(* IEC 61131-3 sources: vertical-injection-machine-docs/docs/IM_SYS_PRG/Code/IO管理/数字量输入, 3 files *)

(* ---- FB_PLCDigitalInputBinder.st ---- *)
(*
  FB_PLCDigitalInputBinder 功能块
  功能：
  1. 把 PLC 运行时输入映像 `IN[0..47]` 刷新到原始 IO 边界 `ST_PLCIO.X*`。
  2. 当前块只负责“采集现场原始数字量输入”，不直接转换为 `ST_MachineSensor`、`ST_PanelIO` 或其他工艺语义。
  3. 当前输入点位顺序固定按现场 IO 表绑定，若现场扩点或换点，必须同步修改本块和 `ST_PLCIO`。

  使用限制：
  1. 当前实现假定目标 PLC 运行时直接提供 `IN[]` 输入映像数组。
  2. 本块应在 `PRG_MainControl` 每拍最前段调用，确保后续逻辑消费到的是本拍最新原始输入。
*)
FUNCTION_BLOCK FB_PLCDigitalInputBinder
VAR_IN_OUT
    stPLC: ST_PLCIO; // 原始 PLC IO 共享边界；本块把现场 `IN[]` 输入映像逐点刷新到其中的 `X*` 字段。
END_VAR

stPLC.X0 := IN[0];      // 把 `IN[0]` 刷新到 `X0`，表示紧急回升原始输入。
stPLC.X1 := IN[1];      // 把 `IN[1]` 刷新到 `X1`，表示低压合模原始输入。
stPLC.X2 := IN[2];      // 把 `IN[2]` 刷新到 `X2`，表示高压合模原始输入。
stPLC.X3 := IN[3];      // 把 `IN[3]` 刷新到 `X3`，表示合模停止原始输入。
stPLC.X4 := IN[4];      // 把 `IN[4]` 刷新到 `X4`，表示电眼输入原始输入。
stPLC.X5 := IN[5];      // 把 `IN[5]` 刷新到 `X5`，表示储料停止原始输入。
stPLC.X6 := IN[6];      // 把 `IN[6]` 刷新到 `X6`，表示拉带停原始输入。
stPLC.X7 := IN[7];      // 把 `IN[7]` 刷新到 `X7`，表示拉带慢速原始输入。
stPLC.X10 := IN[8];     // 把 `IN[8]` 刷新到 `X10`，表示左合模原始输入。
stPLC.X11 := IN[9];     // 把 `IN[9]` 刷新到 `X11`，表示右合模原始输入。
stPLC.X12 := IN[10];    // 把 `IN[10]` 刷新到 `X12`，表示开模停止原始输入。
stPLC.X13 := IN[11];    // 把 `IN[11]` 刷新到 `X13`，表示左托进停原始输入。
stPLC.X14 := IN[12];    // 把 `IN[12]` 刷新到 `X14`，表示左托退停原始输入。
stPLC.X15 := IN[13];    // 把 `IN[13]` 刷新到 `X15`，表示倒带停原始输入。
stPLC.X16 := IN[14];    // 把 `IN[14]` 刷新到 `X16`，表示跳带停原始输入。
stPLC.X17 := IN[15];    // 把 `IN[15]` 刷新到 `X17`，表示二级射出原始输入。
stPLC.X20 := IN[16];    // 把 `IN[16]` 刷新到 `X20`，表示右托进停原始输入。
stPLC.X21 := IN[17];    // 把 `IN[17]` 刷新到 `X21`，表示右托退停原始输入。
stPLC.X22 := IN[18];    // 把 `IN[18]` 刷新到 `X22`，表示座退停止原始输入。
stPLC.X23 := IN[19];    // 把 `IN[19]` 刷新到 `X23`，表示座进停止原始输入。
stPLC.X24 := IN[20];    // 把 `IN[20]` 刷新到 `X24`，表示三级射出原始输入。
stPLC.X25 := IN[21];    // 把 `IN[21]` 刷新到 `X25`，表示中子进停原始输入。
stPLC.X26 := IN[22];    // 把 `IN[22]` 刷新到 `X26`，表示中子退停原始输入。
stPLC.X27 := IN[23];    // 把 `IN[23]` 刷新到 `X27`，表示马达故障原始输入。
stPLC.X30 := IN[24];    // 把 `IN[24]` 刷新到 `X30`，表示安全门原始输入。
stPLC.X31 := IN[25];    // 把 `IN[25]` 刷新到 `X31`，表示模具区域原始输入。
stPLC.X32 := IN[26];    // 把 `IN[26]` 刷新到 `X32`，表示机械手合模原始输入。
stPLC.X33 := IN[27];    // 把 `IN[27]` 刷新到 `X33`，表示机械手托模原始输入。
stPLC.X34 := IN[28];    // 把 `IN[28]` 刷新到 `X34`，表示备用原始输入。
stPLC.X35 := IN[29];    // 把 `IN[29]` 刷新到 `X35`，表示备用原始输入。
stPLC.X36 := IN[30];    // 把 `IN[30]` 刷新到 `X36`，表示射出停止原始输入。
stPLC.X37 := IN[31];    // 把 `IN[31]` 刷新到 `X37`，表示备用原始输入。
stPLC.X40 := IN[32];    // 把 `IN[32]` 刷新到 `X40`，表示备用原始输入。
stPLC.X41 := IN[33];    // 把 `IN[33]` 刷新到 `X41`，表示备用原始输入。
stPLC.X42 := IN[34];    // 把 `IN[34]` 刷新到 `X42`，表示备用原始输入。
stPLC.X43 := IN[35];    // 把 `IN[35]` 刷新到 `X43`，表示备用原始输入。
stPLC.X44 := IN[36];    // 把 `IN[36]` 刷新到 `X44`，表示备用原始输入。
stPLC.X45 := IN[37];    // 把 `IN[37]` 刷新到 `X45`，表示备用原始输入。
stPLC.X46 := IN[38];    // 把 `IN[38]` 刷新到 `X46`，表示备用原始输入。
stPLC.X47 := IN[39];    // 把 `IN[39]` 刷新到 `X47`，表示备用原始输入。
stPLC.X50 := IN[40];    // 把 `IN[40]` 刷新到 `X50`，当前暂定表示启动命令原始输入。
stPLC.X51 := IN[41];    // 把 `IN[41]` 刷新到 `X51`，当前暂定表示停止命令原始输入。
stPLC.X52 := IN[42];    // 把 `IN[42]` 刷新到 `X52`，当前暂定表示复位命令原始输入。
stPLC.X53 := IN[43];    // 把 `IN[43]` 刷新到 `X53`，当前暂定表示急停命令原始输入。
stPLC.X54 := IN[44];    // 把 `IN[44]` 刷新到 `X54`，表示备用原始输入。
stPLC.X55 := IN[45];    // 把 `IN[45]` 刷新到 `X55`，表示备用原始输入。
stPLC.X56 := IN[46];    // 把 `IN[46]` 刷新到 `X56`，表示备用原始输入。
stPLC.X57 := IN[47];    // 把 `IN[47]` 刷新到 `X57`，表示备用原始输入。
END_FUNCTION_BLOCK

(* ---- FB_PLCMachineCommandMapper.st ---- *)
(*
  FB_PLCMachineCommandMapper 功能块
  功能：
  1. 把原始 PLC 数字量输入边界 `ST_PLCIO` 中已经明确语义的公共运行命令点位，翻译为独立机器命令源 `ST_MachineCommand`。
  2. 当前版本只负责 4 个公共运行命令：启动、停止、复位、急停。
  3. 机器模式和手动点动命令仍由面板命令源负责，本块不参与这些字段。

  当前暂定真实来源：
  1. `X50 -> bStart`
  2. `X51 -> bStop`
  3. `X52 -> bReset`
  4. `X53 -> bEStop`

  维护要求：
  1. 若现场后续调整这 4 个命令的真实物理点位，只允许修改本块以及 `PLCIOTypes.st`、`FB_PLCDigitalInputBinder.st` 中对应点位的注释，不要在顶层程序或主控块散写硬编码点号。
  2. 若后续增加 HMI、远程或调试命令源，应新增独立命令源并在 `FB_CommandArbiter` 中继续显式写出优先级。
*)
FUNCTION_BLOCK FB_PLCMachineCommandMapper
VAR_IN_OUT
    stPLC: ST_PLCIO;                    // 原始 PLC IO 边界；本块只读取其中已经在本拍刷新完成的 `X50..X53` 输入点位。
    stCommandSource: ST_MachineCommand; // PLC 数字量独立命令源；本块把公共运行命令回写到这里，供顶层仲裁块统一消费。
END_VAR

(* 先显式清空本命令源不负责的模式字段，避免旧值残留参与最终模式仲裁。 *)
stCommandSource.uiMachineMode := UINT#0;                               // PLC 数字量命令源当前不负责模式选择，因此每拍固定写回 0。

(* 再把 4 个公共运行命令按当前确认的真实物理点位一一映射到独立命令源。 *)
stCommandSource.bStart := stPLC.X50;                                   // 当前暂定把 `X50` 解释为启动命令真实来源，并回写为公共启动命令。
stCommandSource.bStop := stPLC.X51;                                    // 当前暂定把 `X51` 解释为停止命令真实来源，并回写为公共停止命令。
stCommandSource.bReset := stPLC.X52;                                   // 当前暂定把 `X52` 解释为复位命令真实来源，并回写为公共复位命令。
stCommandSource.bEStop := stPLC.X53;                                   // 当前暂定把 `X53` 解释为急停命令真实来源，并回写为公共急停命令。

(* 最后显式清空本命令源不负责的全部手动命令字段，避免独立命令源残留旧的点动语义。 *)
stCommandSource.stManual.bClampStart := FALSE;                         // PLC 数字量命令源当前不负责合模点动启动，因此每拍固定清零。
stCommandSource.stManual.uiClampMode := UINT#0;                        // PLC 数字量命令源当前不负责合模模式号，因此每拍固定清零。
stCommandSource.stManual.bMoldAdjustStart := FALSE;                    // PLC 数字量命令源当前不负责调模点动启动，因此每拍固定清零。
stCommandSource.stManual.uiMoldAdjustMode := UINT#0;                   // PLC 数字量命令源当前不负责调模模式号，因此每拍固定清零。
stCommandSource.stManual.bNozzleStart := FALSE;                        // PLC 数字量命令源当前不负责座台点动启动，因此每拍固定清零。
stCommandSource.stManual.uiNozzleMode := UINT#0;                       // PLC 数字量命令源当前不负责座台模式号，因此每拍固定清零。
stCommandSource.stManual.bInjectStart := FALSE;                        // PLC 数字量命令源当前不负责射胶点动启动，因此每拍固定清零。
stCommandSource.stManual.uiInjectMode := UINT#0;                       // PLC 数字量命令源当前不负责射胶模式号，因此每拍固定清零。
stCommandSource.stManual.bMeterStart := FALSE;                         // PLC 数字量命令源当前不负责储料点动启动，因此每拍固定清零。
stCommandSource.stManual.bEjectStart := FALSE;                         // PLC 数字量命令源当前不负责基础托模点动启动，因此每拍固定清零。
stCommandSource.stManual.uiEjectMode := UINT#0;                        // PLC 数字量命令源当前不负责基础托模模式号，因此每拍固定清零。
stCommandSource.stManual.bEjectModeStart := FALSE;                     // PLC 数字量命令源当前不负责托模组合模式启动，因此每拍固定清零。
stCommandSource.stManual.uiEjectPatternMode := UINT#0;                 // PLC 数字量命令源当前不负责托模组合模式号，因此每拍固定清零。
stCommandSource.stManual.uiEjectTimes := UINT#0;                       // PLC 数字量命令源当前不负责托模循环次数，因此每拍固定清零。
stCommandSource.stManual.bCoreStart := FALSE;                          // PLC 数字量命令源当前不负责中子点动启动，因此每拍固定清零。
stCommandSource.stManual.uiCoreMode := UINT#0;                         // PLC 数字量命令源当前不负责中子模式号，因此每拍固定清零。
stCommandSource.stManual.bMotorStart := FALSE;                         // PLC 数字量命令源当前不负责马达锁存命令，因此每拍固定清零。
stCommandSource.stManual.bTempStart := FALSE;                          // PLC 数字量命令源当前不负责温控启动命令，因此每拍固定清零。
stCommandSource.stManual.bR0 := FALSE;                                 // PLC 数字量命令源当前不负责人工温控 R0，因此每拍固定清零。
stCommandSource.stManual.bR1 := FALSE;                                 // PLC 数字量命令源当前不负责人工温控 R1，因此每拍固定清零。
stCommandSource.stManual.bR2 := FALSE;                                 // PLC 数字量命令源当前不负责人工温控 R2，因此每拍固定清零。
stCommandSource.stManual.bR3 := FALSE;                                 // PLC 数字量命令源当前不负责人工温控 R3，因此每拍固定清零。
END_FUNCTION_BLOCK

(* ---- FB_PLCMachineInputMapper.st ---- *)
(*
  FB_PLCMachineInputMapper 功能块
  功能：
  1. 把原始 PLC 数字量输入边界 `ST_PLCIO` 翻译为机器级语义传感器边界 `ST_MachineSensor`。
  2. 当前块只负责数字量语义与可由当前 IO 表直接推导出的状态，不直接处理模拟量、电子尺或轴实际反馈。
  3. 统一在顶层调用，避免 `PRG_MainControl` 或 `FB_MachineController` 再直接散写 `gvl_stSensor`。

  说明：
  1. 当前现场 IO 表未提供调模停止、射退停止、电子尺与压力尺等独立点位，因此这些字段暂不在本块内改写。
  2. 顶层若后续接入模拟量采集层，应让模拟量采集层在本块之后继续回写 `stSensor` 的相关数值字段。
*)
FUNCTION_BLOCK FB_PLCMachineInputMapper
VAR_IN_OUT
    stPLC: ST_PLCIO;                 // 原始 PLC IO 边界；本块读取其中最新 `X*` 与必要的 `Y36` 状态来生成机器语义输入。
    stSensor: ST_MachineSensor;      // 机器级语义传感器边界；本块负责把当前 IO 表可直接表达的数字量语义统一回写到这里。
END_VAR

(* 先把当前 IO 表中可以直接确定的整机基础条件翻译为机器语义。 *)
stSensor.bDoorClosed := stPLC.X30;                               // 当前先把 `X30` 直接解释为安全门已关语义，供自动准备条件统一使用。
stSensor.bHydReady := stPLC.Y36 AND (NOT stPLC.X27);             // 当前把马达输出镜像与马达故障组合为液压就绪语义；这会相对当前拍命令存在 1 拍延迟，但能保持原始 IO 与机器语义一致。
stSensor.bSystemNoAlarm := NOT stPLC.X27;                        // 当前 IO 表里唯一明确的系统级报警输入是马达故障，因此先用 `NOT X27` 作为系统无报警语义。

(* 再把合模相关停止与到位输入翻译为主控可直接消费的过程语义。 *)
stSensor.bOpenStop := stPLC.X12;                                 // 把 `X12` 翻译为开模停止语义，供合模块按停止信号完成开模段。
stSensor.bCloseLowPres := stPLC.X1;                              // 把 `X1` 翻译为低压合模到位语义，供合模块决定何时切入高压锁模。
stSensor.bCloseHighPres := stPLC.X2;                             // 把 `X2` 翻译为高压合模到位语义，供合模块在按停止/到位模式下结束锁模。
stSensor.bCloseStop := stPLC.X3;                                 // 把 `X3` 翻译为合模停止语义，供合模块在调试和结束模式下统一判断停止。

(* 调模当前缺少独立输入点位，因此先显式保留为 FALSE，避免旧值残留。 *)
stSensor.bMoldAdjustInStop := FALSE;                             // 当前 IO 表未提供独立调模进停止输入，因此本拍明确回写 FALSE。
stSensor.bMoldAdjustOutStop := FALSE;                            // 当前 IO 表未提供独立调模退停止输入，因此本拍明确回写 FALSE。

(* 座台相关停止输入可直接由当前 IO 表表达。 *)
stSensor.bNozzleInStop := stPLC.X23;                             // 把 `X23` 翻译为座进停止语义，供座台模块按停止模式完成座进。
stSensor.bNozzleOutStop := stPLC.X22;                            // 把 `X22` 翻译为座退停止语义，供座台模块按停止模式完成座退。

(* 射胶与储料相关输入按当前 IO 表中已明确的停止点位回写。 *)
stSensor.bInjSeg1Stop := stPLC.X36;                              // 把 `X36` 翻译为一级射出停止语义，供射胶模块在第一段停止模式下结束当前段。
stSensor.bInjSeg2Stop := stPLC.X17;                              // 把 `X17` 翻译为二级射出停止语义，供射胶模块在第二段停止模式下结束当前段。
stSensor.bInjStop := stPLC.X24;                                  // 把 `X24` 翻译为后续射出停止语义，供第三段及以后射出段结束使用。
stSensor.bSuckBackStop := FALSE;                                 // 当前 IO 表未提供独立射退停止输入，因此本拍明确回写 FALSE。
stSensor.bMeterStop := stPLC.X5;                                 // 把 `X5` 翻译为储料停止语义，供储料模块按停止模式推进下一段。

(* 托模当前存在左右两侧停止点；现阶段先按“任一侧命中即视为对应方向到位”翻译语义，避免未装双侧传感器的现场被卡住。 *)
stSensor.bEjectInStop := stPLC.X13 OR stPLC.X20;                 // 把左右托模进停止输入按 OR 汇总为托模进停止语义，供基础托模与托模模式统一消费。
stSensor.bEjectOutStop := stPLC.X14 OR stPLC.X21;                // 把左右托模退停止输入按 OR 汇总为托模退停止语义，供基础托模与托模模式统一消费。

(* 中子进退停止点可以直接由当前 IO 表表达。 *)
stSensor.bCoreInStop := stPLC.X25;                               // 把 `X25` 翻译为中子进停止语义，供中子模块按停止模式结束中子进动作。
stSensor.bCoreOutStop := stPLC.X26;                              // 把 `X26` 翻译为中子退停止语义，供中子模块按停止模式结束中子退动作。
END_FUNCTION_BLOCK
